// SIMATIC S7-200 project (STEP 7-Micro/WIN), CPU 221 REL 01.10

SYMBOL_TABLE USUARIO1
B1               I0.0     // Sensor que detecta entrada de vehículo (NA)
B2               I0.1     // Sensor que detecta salida de vehículo (NA)
S1               I0.2     // Switch final de carrera puerta de entrada cerrada (NA)
S2               I0.3     // Switch final de carrera puerta de entrada abierta (NA)
S3               I0.4     // Switch final de carrera puerta de salida cerrada (NA)
S4               I0.5     // Switch final de carrera puerta de salida abierta (NA)
RESET            I0.6     // Botón pulsador para resetear contador (NA)
M1_ABRE          Q0.0     // Abrir puerta de entrada
M1_CIERRA        Q0.1     // Cerrar puerta de entrada
M2_ABRE          Q0.2     // Abrir puerta de salida
M2_CIERRA        Q0.3     // Cerrar puerta de salida
LIBRE            Q0.4     // Señalización que indica que hay al menos un lugar disponible
LLENO            Q0.5     // Señalización que indica que el estacionamiento está lleno
CARRO1           Q0.6     // Señalización que indica que el lugar 1 esta ocupado
CARRO2           Q0.7     // Señalización que indica que el lugar 2esta ocupado
CARRO3           Q1.0     // Señalización que indica que el lugar 3 esta ocupado
CARRO4           Q1.1     // Señalización que indica que el lugar 4esta ocupado
CARRO5           Q1.2     // Señalización que indica que el lugar 5esta ocupado
CARRO6           Q1.3     // Señalización que indica que el lugar 6 esta ocupado
DISPLAY1         Q2.0     // Display que indica el número de lugares disponibles (BCD).
DISPLAY2         Q2.1     // Display que indica el número de lugares disponibles (BCD).
DISPLAY3         Q2.2     // Display que indica el número de lugares disponibles (BCD).
DISPLAY4         Q2.3     // Display que indica el número de lugares disponibles (BCD).
END_SYMBOL_TABLE

ORGANIZATION_BLOCK PRINCIPAL:OB1
TITLE=COMENTARIOS DEL PROGRAMA
BEGIN
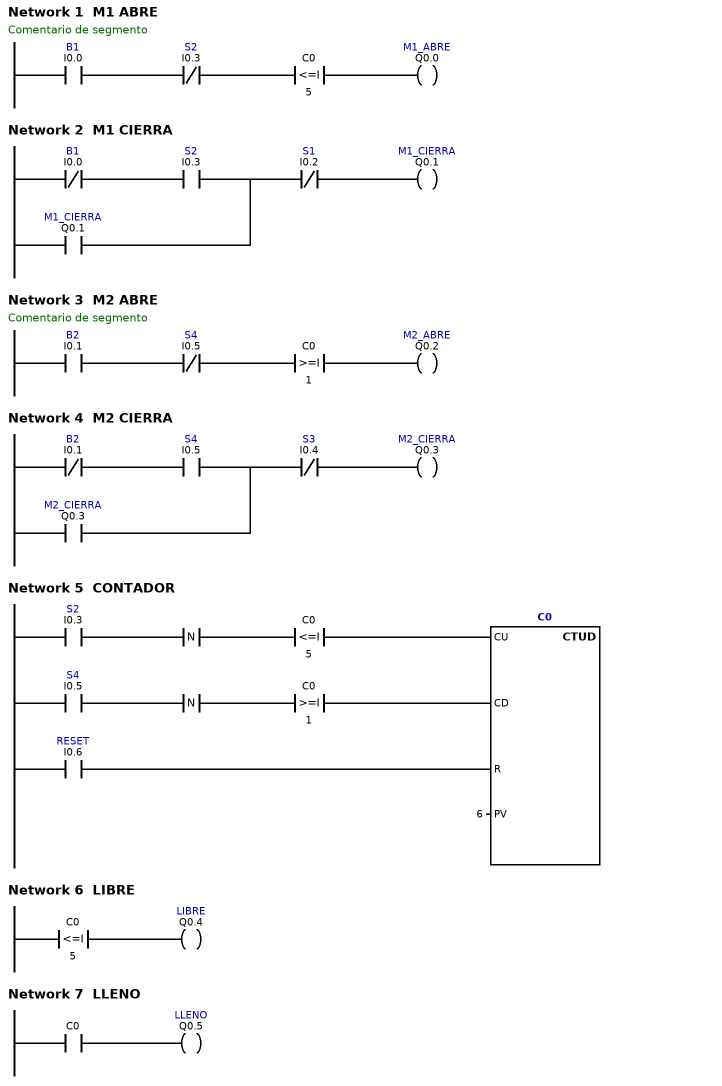
Network 1 // M1 ABRE
// Comentario de segmento
LD     B1:I0.0
AN     S2:I0.3
AW<=   C0, 5
=      M1_ABRE:Q0.0
Network 2 // M1 CIERRA
LDN    B1:I0.0
A      S2:I0.3
O      M1_CIERRA:Q0.1
AN     S1:I0.2
=      M1_CIERRA:Q0.1
Network 3 // M2 ABRE
// Comentario de segmento
LD     B2:I0.1
AN     S4:I0.5
AW>=   C0, 1
=      M2_ABRE:Q0.2
Network 4 // M2 CIERRA
LDN    B2:I0.1
A      S4:I0.5
O      M2_CIERRA:Q0.3
AN     S3:I0.4
=      M2_CIERRA:Q0.3
Network 5 // CONTADOR
LD     S2:I0.3
ED
AW<=   C0, 5
LD     S4:I0.5
ED
AW>=   C0, 1
LD     RESET:I0.6
CTUD   C0, 6
Network 6 // LIBRE
LDW<=  C0, 5
=      LIBRE:Q0.4
Network 7 // LLENO
LD     C0
=      LLENO:Q0.5
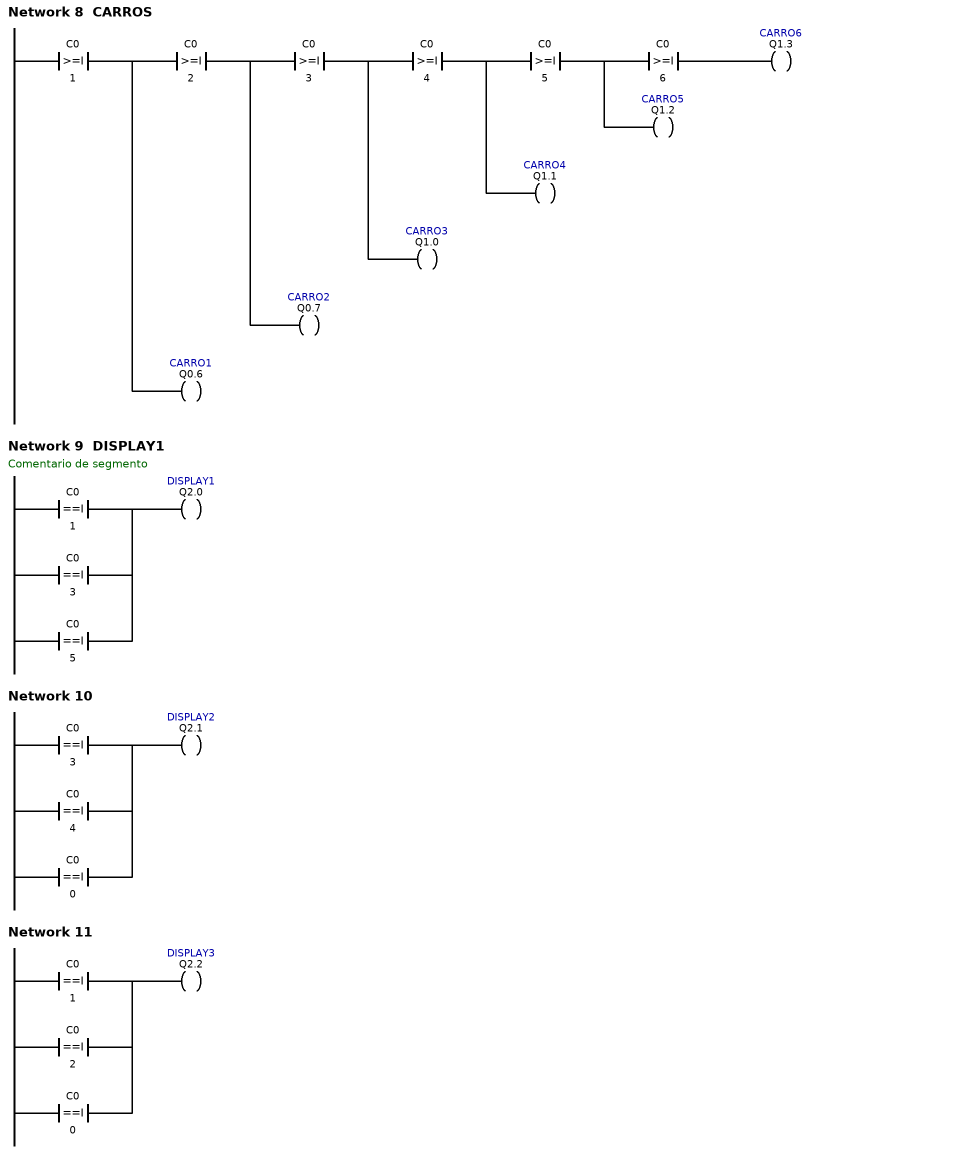
Network 8 // CARROS
LDW>=  C0, 1
LPS
AW>=   C0, 2
LPS
AW>=   C0, 3
LPS
AW>=   C0, 4
LPS
AW>=   C0, 5
LPS
AW>=   C0, 6
=      CARRO6:Q1.3
LPP
=      CARRO5:Q1.2
LPP
=      CARRO4:Q1.1
LPP
=      CARRO3:Q1.0
LPP
=      CARRO2:Q0.7
LPP
=      CARRO1:Q0.6
Network 9 // DISPLAY1
// Comentario de segmento
LDW=   C0, 1
OW=    C0, 3
OW=    C0, 5
=      DISPLAY1:Q2.0
Network 10
LDW=   C0, 3
OW=    C0, 4
OW=    C0, 0
=      DISPLAY2:Q2.1
Network 11
LDW=   C0, 1
OW=    C0, 2
OW=    C0, 0
=      DISPLAY3:Q2.2
END_ORGANIZATION_BLOCK
